TYPE T_AnyNum : __SYSTEM.AnyType; END_TYPE

(* stored: Version 1.1.0.1
   DUT T_AnyNum: Id {0251880a-807f-49ff-a784-bd877de388d2} *)
